PROGRAM prgLightSwitch
VAR
	fbLight : FB_Light;
	bSwitchOn : BOOL; //{#lynus.ag#()}
	bSwitchOff : BOOL; //{#lynus.ag#()}
	bStateLight : BOOL; //{#lynus.ag#()}
END_VAR

fbLight(bOn:=bSwitchOn, bOff:=bSwitchOff, bLight=>bStateLight);

END_PROGRAM

(* stored: Version 1.1.0.1, ProductVersion 3.1.4024.11
   POU prgLightSwitch: Id {81341900-eb74-404d-8e3c-ae2de52a0211}, SpecialFunc None *)
